Universal Robots PolyScope program: xmlrpc_deteccion_fresas_vertical_pinza_v2.urp

Program xmlrpc_deteccion_fresas_vertical_pinza_v2 (installation=deteccion directory=/programs/usbdisk/Versiones xmlrpc_deteccion_fresas createdIn=5.17.0 lastSavedIn=5.21.0 robotSerialNumber=20215500624)
Calibrated DH parameters: a=[0.000186, -0.025908, -0.392311, -0.000071, 0.00009, 0]; d=[0.162736, -361.104072, 360.092318, 1.145413, 0.099738, 0.099626]; alpha=[1.57079, -0.001175, 0.009075, 1.569386, -1.569463, 0]; deltaTheta=[0, 1.509811, 4.749978, 0.023394, 0, -0.000001]
InitVariablesNode
BeforeStart
  Folder Configuracion XMLRPC
    'Configuración del XMLRPC'
    camera := rpc_factory("xmlrpc","http://192.168.23.107:50000")
  Folder Inicializacion variables
    'Variable para ver si se detecta dos veces el mismo pto'
    next_pose_aux := p[0,0,0,0,0,0]
  Folder Centro coord camara
    'Punto de referencia de la camara (centro de coordenadas camara)'
    SuppressedNode
      MoveJ speed 60 deg/s, acceleration 80 deg/s^2 (useActiveTCP=true optimoveEnabled=false optiMoveSpeed=0.3 optiMoveAcceleration=0.09) feature=Plano_camara
        Waypoint reference_p: TCP in base x=-205.136 y=303.641 z=-13.102 mm, rx=-1.1967 ry=-2.9046 rz=-0.0001 rad; joints [-215.195, -141.895, -109.787, -18.283, 89.252, -81.03] deg; TCP offset x=0 y=0 z=20 mm, rx=0 ry=0 rz=0 rad; feature pose in base x=-205.136 y=303.641 z=-13.102 mm, rx=-1.1967 ry=-2.9046 rz=-0.0001 rad
  Folder Inicializacion pinza
    URCap Liberación 2FG (OnRobot, OnRobot A/S) dataModel(twofg.target-speed=60, twofg.external-grip.target-width=0.0705999984741211, twofg.internal-grip.target-width=0.0845999984741211)
    SuppressedNode
      URCap Agarre 2FG (OnRobot, OnRobot A/S) dataModel(twofg.target-speed=91, external_internal_action.index=0, twofg.target-force=50, workpiece-lost=true, twofg.internal-grip.target-width=0.013, twofg.external-grip.target-width=0.0)
Robot Program (runOnlyOnce=false)
  Folder Home
    'Home: Punto inicial para posterior recogida de deteccion'
    MoveJ speed 60 deg/s, acceleration 80 deg/s^2 (useActiveTCP=true optimoveEnabled=true optiMoveSpeed=0.21 optiMoveAcceleration=0.044) feature=Plano_pared
      Waypoint Casa: TCP in base x=-257.547 y=-358.533 z=297.396 mm, rx=-0.045 ry=-2.1837 rz=2.2158 rad; joints [-3.35, -97.855, 155.633, -173.043, 1.173, -64.771] deg; TCP offset x=0 y=0 z=138.6 mm, rx=0 ry=0 rz=0 rad; feature pose in base x=-499.77 y=-438.077 z=375.606 mm, rx=0.0174 ry=2.1723 rz=-2.2092 rad
  Folder Comunicacion camara
    'Obtencion de datos de la camara'
    next_pose := camera.get_next_pose()
    'Se hace el cambio de unidades mm a m'
    next_pose_list := p[next_pose[0]/1000,next_pose[1]/1000,0,0,0,0]
  Folder Movimiento UR
    If next_pose_list[0]≟0  and next_pose_list[1]≟0
      Folder NO_Deteccion
        MoveJ speed 60 deg/s, acceleration 80 deg/s^2 (useActiveTCP=true optimoveEnabled=false optiMoveSpeed=0.3 optiMoveAcceleration=0.09) feature=Plano_pared
          Waypoint Casa: TCP in base x=-257.547 y=-358.533 z=297.396 mm, rx=-0.045 ry=-2.1837 rz=2.2158 rad; joints [-3.35, -97.855, 155.633, -173.043, 1.173, -64.771] deg
    Else 
      Folder Deteccion_OK
        If next_pose_aux ≠ next_pose_list
          'Hay detecciones que recoger'
          'Posicion de la recogida'
          MoveL speed 250 mm/s, acceleration 1200 mm/s^2 (useActiveTCP=true optimoveEnabled=false optiMoveSpeed=0.3 optiMoveAcceleration=0.09) feature=Plano_pared
            Waypoint Variable (Variable): variable=next_pose_list
            SuppressedNode
              Waypoint Pick_fresa: TCP in base x=-437.129 y=-443.32 z=438.117 mm, rx=0.0174 ry=2.1723 rz=-2.2092 rad; joints [9.082, -81.552, 88.882, -17.685, 7.985, -167.498] deg
            SuppressedNode
              Waypoint Salida_pick: TCP in base x=-437.895 y=-408.891 z=437.523 mm, rx=0.0174 ry=2.1723 rz=-2.2092 rad; joints [4.823, -85.723, 94.442, -30.343, 3.889, -156.203] deg
            SuppressedNode
              URCap Agarre 2FG (OnRobot, OnRobot A/S)
          'Variable aux para comparar listas '
          next_pose_aux := p[next_pose_list[0],next_pose_list[1],next_pose_list[2],0,0,0]
        Else 
          'No hay detecciones que recoger'
          MoveJ speed 60 deg/s, acceleration 80 deg/s^2 (useActiveTCP=true optimoveEnabled=false optiMoveSpeed=0.3 optiMoveAcceleration=0.09) feature=Plano_pared
            Waypoint Casa: TCP in base x=-257.547 y=-358.533 z=297.396 mm, rx=-0.045 ry=-2.1837 rz=2.2158 rad; joints [-3.35, -97.855, 155.633, -173.043, 1.173, -64.771] deg
  Wait Sleep waitTime=1
